FUNCTION_BLOCK fbSignalSimXYMover
VAR_IN_OUT
	em : ST_EM;
END_VAR
VAR_INPUT
	EnableSim : BOOL;
	CmdSim : BOOL := true;
END_VAR
VAR
	TimerSim : Array[1..10] OF TON;
	Elapsed : TIME;
END_VAR

IF EnableSim THEN
	CASE em.SequenceStep OF
		
	1: 	TimerSim[1](in := TRUE);
		TimerSim[1](PT := T#2S);
		
		IF TimerSim[1].Q THEN
			em.Config.Data.I[1] := FALSE;
            em.Config.Data.I[2] := FALSE;
            em.Config.Data.I[3] := FALSE;
            em.Config.Data.I[4] := FALSE;
			TimerSim[1](in := FALSE);
		END_IF
		
	3: 	TimerSim[2](in := TRUE);
		TimerSim[2](PT := T#2S);
		
		IF TimerSim[2].Q THEN
			em.Config.Data.I[1] := TRUE;
            em.Config.Data.I[3] := TRUE;
			em.Cmd := E_CMD.reset;
			TimerSim[2](in := FALSE);
		END_IF
	
		
	5: 	TimerSim[3](in := TRUE);
		TimerSim[3](PT := T#2S);
		
		IF TimerSim[3].Q THEN
			em.Config.Data.I[1] := FALSE;
            em.Config.Data.I[2] := FALSE;
            em.Config.Data.I[3] := FALSE;
            em.Config.Data.I[4] := FALSE;
			TimerSim[3](in := FALSE);
		END_IF
	
	6:	TimerSim[4](in := TRUE);
		TimerSim[4](PT := T#2S);
		
		IF TimerSim[4].Q THEN
			em.Cmd := E_CMD.clear;
			TimerSim[4](in := FALSE);
		END_IF
	
	10: TimerSim[5](in := TRUE);
		TimerSim[5](PT := T#2S);
		
		IF TimerSim[5].Q THEN
			em.Cmd := E_CMD.start;
			TimerSim[5](in := FALSE);
		END_IF
		
	
	20:	TimerSim[6](in := TRUE);
		TimerSim[6](PT := T#2S);
		
		IF TimerSim[6].Q THEN
			em.Config.Data.I[5] := TRUE;
			TimerSim[6](in := FALSE);
		END_IF
		
	30: TimerSim[7](in := TRUE);
		TimerSim[7](PT := T#2S);
		
		IF TimerSim[7].Q THEN
			em.Config.Data.I[1] := FALSE;
			em.Config.Data.I[2] := TRUE;
			TimerSim[7](in := FALSE);
		END_IF
	
	40: TimerSim[8](in := TRUE);
		TimerSim[8](PT := T#2S);
		
		IF TimerSim[8].Q THEN
			em.Config.Data.I[3] := FALSE;
			em.Config.Data.I[4] := TRUE;
			TimerSim[8](in := FALSE);
		END_IF

		
	60:	TimerSim[9](in := TRUE);
		TimerSim[9](PT := T#2S);
		
		IF TimerSim[9].Q THEN
			em.Config.Data.I[5] := FALSE;
			TimerSim[9](in := FALSE);
		END_IF
	
	70: TimerSim[10](in := TRUE);
		TimerSim[10](PT := T#2S);
		
		IF TimerSim[9].Q THEN
			em.Config.Data.I[1] := TRUE;
			em.Config.Data.I[3] := TRUE;
			TimerSim[9](in := FALSE);
		END_IF
	
	
	END_CASE 
END_IF

END_FUNCTION_BLOCK

(* stored: Version 1.1.0.1, ProductVersion 3.1.4024.12
   POU fbSignalSimXYMover: Id {7169e8eb-476f-4bb5-9ffe-cfa494d7f0fc}, SpecialFunc None *)
